// SIMATIC STEP 7 (V5.x) project UNDODERALEX
// CPU: CPU 314C-2 DP
// station: Hardware
// station: SIMATIC 300(1)
// station: P_ADR_BUS
// program: S7-Programm(2)

SYMBOL_TABLE
"UNDODER"	FC 1	FC 1
"Zyklus"	OB 1	OB 1
END_SYMBOL_TABLE

FUNCTION "UNDODER" : VOID	// FC 1
VERSION : 0.1
BEGIN
NETWORK
TITLE =
// (network holds code this reader does not know; not shown)
NETWORK
TITLE =
//rot
// (network holds code this reader does not know; not shown)
NETWORK
TITLE =
//rot/gelb: rot
// (network holds code this reader does not know; not shown)
NETWORK
TITLE =
//rot/gelb: gelb
NETWORK
TITLE =
//grün
NETWORK
TITLE =
//gelb only (5)
//
NETWORK
TITLE =
//grün blink
// (network holds code this reader does not know; not shown)
END_FUNCTION

ORGANIZATION_BLOCK "Zyklus"	// OB 1
TITLE = "Main Program Sweep (Cycle)"
VERSION : 0.1
VAR_TEMP
  OB1_EV_CLASS : BYTE ;	//Bits 0-3 = 1 (Coming event), Bits 4-7 = 1 (Event class 1)
  OB1_SCAN_1 : BYTE ;	//1 (Cold restart scan 1 of OB 1), 3 (Scan 2-n of OB 1)
  OB1_PRIORITY : BYTE ;	//Priority of OB Execution
  OB1_OB_NUMBR : BYTE ;	//1 (Organization block 1, OB1)
  OB1_RESERVED_1 : BYTE ;	//Reserved for system
  OB1_RESERVED_2 : BYTE ;	//Reserved for system
  OB1_PREV_CYCLE : INT ;	//Cycle time of previous OB1 scan (milliseconds)
  OB1_MIN_CYCLE : INT ;	//Minimum cycle time of OB1 (milliseconds)
  OB1_MAX_CYCLE : INT ;	//Maximum cycle time of OB1 (milliseconds)
  OB1_DATE_TIME : DATE_AND_TIME ;	//Date and time OB1 started
END_VAR
BEGIN
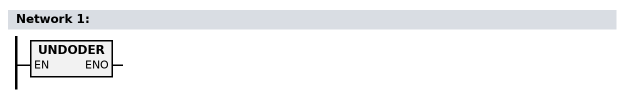
NETWORK
TITLE =
      CALL  "UNDODER";
      NOP   0;
END_ORGANIZATION_BLOCK
